Fanuc KAREL source: kt00272.KL

-- PROVISIONAL review KL for V1013-1; original PC SHA256 e2df323528f3874c165e1804725aabc3dccbc98801013c23cd35e7a9ae69ca66
-- Incomplete behavior may be omitted. Consult companion uncertainty JSON. Do not deploy.
PROGRAM KT00272
%NOLOCKGROUP
VAR
  R2 : REAL
  OUT : BOOLEAN
-- UNRESOLVED_DECL H1 type=002017
BEGIN
  -- UNRESOLVED_PC offsets 5-19; opcodes 2E,22,9D,33,B4
  -- UNRESOLVED_PC offsets 24-35; opcodes 2E,23
  -- UNRESOLVED_PC offsets 40-64; opcodes 22,9D,33,B3,21,29,64,6D,23
  -- UNRESOLVED_PC offsets 69-73; opcodes 7F
END KT00272
